// Fluent builder interface for composing log entries.
// Obtain an instance via F_Log() or FB_Log.Log(), chain methods, and call CreateLog() to emit.
INTERFACE I_WithLogger EXTENDS I_Logger

// Overrides the default logger name for this log entry.
// If not called, the global logger or FB_Log instance logger is used.
METHOD WithLogger : I_WithContext
VAR_INPUT
	sLogger	: T_MaxString;
END_VAR
END_METHOD

END_INTERFACE

(* stored: Version 1.1.0.1, ProductVersion 3.1.4026.18
   Itf I_WithLogger: Id {37a6dead-b272-0175-2d5c-85a4173fe999}
   Method WithLogger: Id {3aba0bb2-12cb-0edb-2d3d-6cff8af1a20d} *)
